# B&R Automation Studio project 305841_E00002_0 (part 5)

#### ActionMotionFbs.st
```iecst
(********************************************************************
 * COPYRIGHT -- General Atomics
 ********************************************************************
 * Program: AxisStateMachine
 * File: ActionMoveVel.st
 * Author: Administrator
 * Created: January 22, 2014
 ********************************************************************
 * Implementation of program AxisStateMachine
 ********************************************************************)

ACTION ActionCallMotionFunctions:
  ActionRangeCheckMoveParams;
  ActionMpAxisBasic;
  ActionReadDrivePos;
  ActionCamInOut;
  ActionGearInOut;
  ActionOffsetShift;
  ActionPhaseShift;
END_ACTION

ACTION ActionRangeCheckMoveParams:
  // Range checks position, velocity, accel & Decel

  // Make sure min/max values are not exceeded for position, velocity, accel, and decel.
  // Clamp if necessary.

  // Position
  ax.MoveParameters.Position := MIN(axPositionLimits.PositionLimitPos, MAX(axPositionLimits.PositionLimitNeg, ax.MoveParameters.Position));

  // Velocity
  ax.MoveParameters.Velocity := MIN(ax.MoveParameters.VelocityMax, MAX(ax.MoveParameters.VelocityMin, ax.MoveParameters.Velocity));

  // Accel and decel
  ax.MoveParameters.Acceleration := MIN(ax.MoveParameters.AccelMax, MAX(ax.MoveParameters.AccelMin, ax.MoveParameters.Acceleration));
  ax.MoveParameters.Deceleration := MIN(ax.MoveParameters.DecelMax, MAX(ax.MoveParameters.DecelMin, ax.MoveParameters.Deceleration));

END_ACTION

ACTION ActionMpAxisBasic:
  // 1) Assume velocity, accel & Decel have been range checked
  // 2) Packs the sMot_MoveParameters into a local axisBasicParamsStructure
  // 3) Detects parameter changes and manages the Update and UpdateDone bits
  // 4) Sets the fb command bits based on the axis sMot_AxisCommands structure
  // 5) Runs the fbMpAxisBasic funciton block
  // 6) Updates the axis structure with the status and axis info coming back from the fb

  // The execution behavior is determined by the inputs set elsewhere
  // in particular the sMot_AxisCommands XxxxCmd bits,
  // and the values in sMot_MoveParameters structure

  // Axis reference set in init routine

  // Only enable the fb if the axis is not set to be ignored
  // TODO: Different check needed? Not sure how to tell if an axis reference is not set
  // It would be nice to check ax.fbMpAxisBasic.MpLink <> 0 for example, but this is a structure not an address
  IF NOT ax.Ignore AND ax.AxisNo <> 0 THEN
    ax.fbMpAxisBasic.Enable := TRUE;
  ELSE
    ax.fbMpAxisBasic.Enable := FALSE;
  END_IF;

  // Load the parameters from the sMot_MoveParameter structure into
  // local structure variables used for the fb
  fctPackMpAxisBasicParams(_I_UdtParams:= ADR(ax.MoveParameters), _IO_MpParams := axisBasicParams);

  // To allow move parameter changes to take effect without having to stop,
  // detect a difference between the desired parameters and the previous values.
  // If they are different, then set the update bit until the UpdateDone bit is set.
  // NOTE: This fb manages the ax.fbMpAxisCoupling.Update request and monitors the .UpdateDone bit
  // Use the .UpdateCouplingParams bit in the command structure if the application needs to control
  // when to trigger the update. If parameters need to be set in possibly different areas of the software,
  // and all the updates should take place at once, the update fb is called conditionally. The
  // checked bit can be set high so it is called all the time if the checked bit is not managed.
  ax.Commands.UpdateMoveParams:= TRUE;
  IF ax.Commands.UpdateMoveParams THEN
    ax.fbUpdateBFbParams(_IO_MpParams := axisBasicParams);
    ax.Commands.UpdateMoveParams := FALSE;
  END_IF;

  // TODO: Enforce move permissives

  // Use the commands from the axis structue
  ax.fbMpAxisBasic.ErrorReset := ax.Commands.DriveResetCmd;
  ax.fbMpAxisBasic.Power := ax.Commands.EnableCmd;
  ax.fbMpAxisBasic.Home := ax.Commands.HomeCmd;
  // There is no specific jog cmd. Use Move Velocity instead.
  ax.fbMpAxisBasic.MoveVelocity := ax.Commands.MoveVelocityCmd OR ax.Commands.MoveJogCmd;
  ax.fbMpAxisBasic.MoveAbsolute := ax.Commands.MoveAbsoluteCmd;
  ax.fbMpAxisBasic.MoveAdditive := ax.Commands.MoveRelativeCmd;
  ax.fbMpAxisBasic.Stop := ax.Commands.StopCmd;
  ax.fbMpAxisBasic.JogPositive := ax.Commands.MoveJogPositiveCmd;
  ax.fbMpAxisBasic.JogNegative := ax.Commands.MoveJogNegativeCmd;
  ax.fbMpAxisBasic.LimitLoad := ax.MoveParameters.EnableTorqueLimit;
  ax.fbMpAxisBasic.ReleaseBrake := ax.Commands.ReleaseBrakeCmd;
  ax.fbMpAxisBasic.AutoTune := FALSE; // TODO
  ax.fbMpAxisBasic.Simulate := FALSE; // TODO

  // Call the fb
  ax.fbMpAxisBasic();

  // Update the axis status structure
  ax.Status.Position := ax.fbMpAxisBasic.Position;
  ax.Status.Velocity := ax.fbMpAxisBasic.Velocity;
  ax.Status.IsPoweredOn := ax.fbMpAxisBasic.PowerOn;
  ax.Status.IsHomed := ax.fbMpAxisBasic.IsHomed;
  ax.Status.IsInVelocity := ax.fbMpAxisBasic.InVelocity;
  ax.Status.IsInPosition := ax.fbMpAxisBasic.InPosition;
  ax.Status.IsMoveActive := ax.fbMpAxisBasic.MoveActive;
  ax.Status.IsMoveDone := ax.fbMpAxisBasic.MoveDone;
  ax.Status.IsStopped := ax.fbMpAxisBasic.Stopped;
  ax.Status.IsTorqueLimitReady := ax.fbMpAxisBasic.LimitLoadReady;
  ax.Status.IsBrakeManuallyReleased := ax.fbMpAxisBasic.BrakeReleased;

  // Now load the sMot_AxisStatus structure with the data returned from the fb
  fctGetMpAxisInfo(_I_MpInfo := ADR(ax.fbMpAxisBasic.Info), _IO_UdtStatus := ax.Status);

  // Calculate special (algorithmic) positions
  CalcSpecialPositions;

  // Now that the status of this axis is known, copy it to the other axes slave status
  // area if this axis is specified as a slave.
  CopySlaveStatusToMaster;

END_ACTION

ACTION ActionReadDrivePos:
  // Read the drive position. As opposed to the position value coming from MpAxisBasic,
  // the drive position allows different position sources to be specified, but it also
  // allows can provide the position that does not have a MOD applied in the periodic case.
  // This is helpful to assess long moves on periodic axes (e.g. 1000 degree move on a
  // 360 degree periodic axis).
  // Only execute the read position fb if the axis number has been set,
  // the axis is not ignored.
  IF NOT ax.Ignore AND ax.AxisNo <> AD_UNKNOWN THEN
    // Axis is in play. Go get some of that position ...
    // Set the source, enable the fb
    ax.fbReadDrivePos.ValueSource := mcVALUE_ACTUAL_AXIS_UNITS;
    ax.fbReadDrivePos.Enable := TRUE;
  ELSE
    // axis should be ignored
    // keep the enable low
    ax.fbReadDrivePos.Enable := FALSE;
  END_IF;

  // Fb should be set up. Call 'er
  ax.fbReadDrivePos();

  // If fb has been enabled and is valid and error , get the drive position. Otherwise
  // use the sentinel value
  IF ax.fbReadDrivePos.Enable AND ax.fbReadDrivePos.Valid AND NOT ax.fbReadDrivePos.Error THEN
    ax.Status.DrivePosition := ax.fbReadDrivePos.CyclicPosition;
  ELSE
    ax.Status.DrivePosition := INVALID_SENTINEL_LREAL;
  END_IF;

END_ACTION

ACTION ActionCamInOut:
  // Execute the cam in or cam out fbs based on the CamIn/Out requests
  // The fbs are edge triggered, and the requests are cleared once serviced.
  // If the caming params change, another request must be made.
  // TODO: Is cam out and another cam in needed if params change?

  // Only execute the cam in fb if the axis number has been set,
  // the slave axis number has been set, and neither is set to be ignored,
  // and it is requested.
  IF ax.Ignore OR ax.AxisNo = AD_UNKNOWN OR
       ax.CouplingParameters.SlaveAxisNo = AD_UNKNOWN OR
       axes[ax.CouplingParameters.SlaveAxisNo].Ignore THEN
    // slave or master should be ignored
    // keep the requests and executes low
    ax.CouplingParameters.CamInReq := FALSE;
    ax.CouplingParameters.CamOutReq := FALSE;
    ax.fbCamIn.Execute := FALSE;
    ax.fbCamOut.Execute := FALSE;
  ELSIF ax.CouplingParameters.CamInReq THEN
    // CamIn request is made.
    // Clear the req so a future rising edge can be seen
    ax.CouplingParameters.CamInReq := FALSE;
    // Make sure the CamOut req and execute is clear
    ax.CouplingParameters.CamOutReq := FALSE;
    ax.fbCamOut.Execute := FALSE;
    // Load the cam in params, then set the execute input (edge triggered fb)
    ax.fbCamIn.MasterOffset := ax.CouplingParameters.CamMasterOffset;
    ax.fbCamIn.SlaveOffset := ax.CouplingParameters.CamSlaveOffset;
    ax.fbCamIn.MasterScaling := ax.CouplingParameters.CamScalingMaster;
    ax.fbCamIn.SlaveScaling := ax.CouplingParameters.CamScalingSlave;
    ax.fbCamIn.StartMode := ax.CouplingParameters.CamStartMode;
    ax.fbCamIn.MasterValueSource := ax.CouplingParameters.CamMasterValueSource;
    ax.fbCamIn.CamID := ax.CouplingParameters.CamId;
    ax.fbCamIn.BufferMode := ax.CouplingParameters.CamBufferMode; // only mcAborting currently supported
    ax.fbCamIn.AdvancedParameters.Periodic := ax.CouplingParameters.CamIsPeriodic;
    ax.fbCamIn.AdvancedParameters.Velocity := 0.0; // disable, use (slave?) axis max vel
    ax.fbCamIn.AdvancedParameters.Acceleration := 0.0; // disable, use (slave?) axis max accel
    ax.fbCamIn.AdvancedParameters.Deceleration := 0.0; // disable, use (slave?) axis max decel
    ax.fbCamIn.AdvancedParameters.Jerk := 0.0; // only non-zero if using McProfGen
    ax.fbCamIn.Execute := TRUE; // fb looks for a rising edge
  ELSIF ax.CouplingParameters.CamOutReq THEN
    // Clear the req so a future rising edge can be seen
    ax.CouplingParameters.CamOutReq := FALSE;
    // Make sure the GearIn req and execute is clear
    ax.CouplingParameters.CamInReq := FALSE;
    ax.fbCamIn.Execute := FALSE;
    // Load the cam out params, then set the execute input (edge triggered fb)
    ax.fbCamOut.Jerk := 0.0; // only non-zero if using McProfGen
    ax.fbCamOut.Execute := TRUE;
  END_IF;

  // Call the cam in and cam out fbs.
  ax.fbCamIn();
  ax.fbCamOut();
  // Clear the exuecute bits. The fbs are edge triggerd, and would have been seen by the above call.
  ax.fbCamIn.Execute := FALSE;
  ax.fbCamOut.Execute := FALSE;

  // Update the axis status structure
  IF NOT ax.fbCamIn.Error THEN
    ax.Status.IsCamInSync := ax.fbCamIn.InSync;
    ax.Status.IsCamEndOfProfile := ax.fbCamIn.EndOfProfile;
    ax.Status.CamStatus := ax.fbCamIn.Status;
  ELSE
    ax.Status.IsCamInSync := FALSE;
    ax.Status.IsCamEndOfProfile := FALSE;
    ax.Status.CamStatus := mcCAM_STATUS_PREPARING_MOVE; // 0 value, but don't have a good choice for "not active"
  END_IF;

END_ACTION

ACTION ActionGearInOut:
  // Execute the gear in or gear out fbs based on the GearIn/Out requests
  // The fbs are edge triggered, and the requests are cleared once serviced.
  // If the gearing params change, another request must be made.

  // Only execute the gear in fb if the axis number has been set,
  // the slave axis number has been set, and neither is set to be ignored,
  // and it is requested.
  IF ax.Ignore OR ax.AxisNo = AD_UNKNOWN OR
       ax.CouplingParameters.SlaveAxisNo = AD_UNKNOWN OR
       axes[ax.CouplingParameters.SlaveAxisNo].Ignore THEN
    // slave or master should be ignored
    // keep the requests and executes low
    ax.CouplingParameters.GearInReq := FALSE;
    ax.CouplingParameters.GearOutReq := FALSE;
    ax.fbGearIn.Execute := FALSE;
    ax.fbGearOut.Execute := FALSE;
  ELSIF ax.CouplingParameters.GearInReq THEN
    // GearIn request is made.
    // Clear the req so a future rising edge can be seen
    ax.CouplingParameters.GearInReq := FALSE;
    // Make sure the GearOut req and execute is clear
    ax.CouplingParameters.GearOutReq := FALSE;
    ax.fbGearOut.Execute := FALSE;
    // Load the gear in params, then set the execute input (edge triggered fb)
    ax.fbGearIn.RatioNumerator := ax.CouplingParameters.GearInRatioNumerator;
    ax.fbGearIn.RatioDenominator := ax.CouplingParameters.GearInRatioDenominator;
    ax.fbGearIn.MasterValueSource := ax.CouplingParameters.GearInMasterValueSource;
    ax.fbGearIn.Acceleration := ax.CouplingParameters.ShiftAccelerationMax;
    ax.fbGearIn.Deceleration := ax.CouplingParameters.ShiftDecelerationMax;
    ax.fbGearIn.Jerk := ax.CouplingParameters.ShiftJerk; // only non-zero if using McProfGen
    ax.fbGearIn.BufferMode := ax.CouplingParameters.GearInBufferMode; // onlly mcAborting currently supported
    ax.fbGearIn.AdvancedParameters.MasterMaxVelocity := ax.CouplingParameters.ShiftProfileBaseMaxVelocity;
    ax.fbGearIn.Execute := TRUE; // fb looks for a rising edge
  ELSIF ax.CouplingParameters.GearOutReq THEN
    // Clear the req so a future rising edge can be seen
    ax.CouplingParameters.GearOutReq := FALSE;
    // Make sure the GearIn req and execute is clear
    ax.CouplingParameters.GearInReq := FALSE;
    ax.fbGearIn.Execute := FALSE;
    // Load the gear out params, then set the execute input (edge triggered fb)
    ax.fbGearOut.Jerk := 0.0; // only non-zero if using McProfGen
    ax.fbGearOut.Execute := TRUE;
  END_IF;

  // Call the gear in and gear out fbs.
  ax.fbGearIn();
  ax.fbGearOut();
  // Clear the exuecute bits. The fbs are edge triggerd, and would have been seen by the above call.
  ax.fbGearIn.Execute := FALSE;
  ax.fbGearOut.Execute := FALSE;

  // Update the axis status structure.
  // Derrive InCompensation -- Active but not in sync
  IF ax.fbGearIn.Active AND NOT ax.fbGearIn.Error THEN
    // If gear in is active, it is either in sync or in compensation
    ax.Status.IsGearInSync := ax.fbGearIn.InGear;
    ax.Status.IsGearInCompensation := NOT ax.fbGearIn.InGear;
  ELSE
    ax.Status.IsGearInSync := FALSE;
    ax.Status.IsGearInCompensation := FALSE;
  END_IF;

END_ACTION

ACTION ActionOffsetShift:
  // Execute the offset shift fb based on the offset shift request.
  // The fb has a level sensitive enable and an edge triggered StartShift input.
  // NOTE: Either by design or because of a bug, the AdvancedParameters.ProfileBase
  // seems to be evaluated based on Enable going high. Changes made to the ProfileBase,
  // after enable going high but before StartShift input going high are ignored.
  // If the shift params change, another request must be made.
  // A shift cannot be stopped once started without halting or some oher means of stopping
  // the axes outside the scope of the shift fb.

  // Since triggering an offset while another shift is in progress triggers an error,
  // the request, enable, and start shift are only cleared once the shift is finished,
  // or the fb is invalid or in error

  // Only execute the offset shift fb if the axis number has been set,
  // the slave axis number has been set, and neither is set to be ignored
  IF ax.Ignore OR ax.AxisNo = AD_UNKNOWN OR
    ax.CouplingParameters.SlaveAxisNo = AD_UNKNOWN OR
    axes[ax.CouplingParameters.SlaveAxisNo].Ignore THEN
    // slave or master should be ignored, or slave is not set, or
    // master is not powered.  Keep the request, enable, and startshift low
    ax.CouplingParameters.OffsetShiftReq := FALSE;
    ax.fbOffsetShift.Enable := FALSE;
    ax.fbOffsetShift.StartShift := FALSE;
  ELSIF ax.CouplingParameters.OffsetShiftReq AND NOT ax.fbOffsetShift.Enable THEN
    // Offset Shift request is made.
    // Set the fb params so a start shift can act on them. Set them
    // before bringing enable high because the profile base param(s) seem to
    // need to be set before the StartShift input is raised.
    ax.fbOffsetShift.OffsetShift := ax.CouplingParameters.Shift;
    ax.fbOffsetShift.Velocity := ax.CouplingParameters.ShiftVelocityMax;
    ax.fbOffsetShift.Acceleration := ax.CouplingParameters.ShiftAccelerationMax;
    ax.fbOffsetShift.AdvancedParameters.ShiftMode := ax.CouplingParameters.ShiftMode;
    ax.fbOffsetShift.AdvancedParameters.ProfileBase := ax.CouplingParameters.ShiftProfileBase;
    ax.fbOffsetShift.AdvancedParameters.ProfileBaseMaxVelocity := ax.CouplingParameters.ShiftProfileBaseMaxVelocity;
    ax.fbOffsetShift.AdvancedParameters.DistanceParameters.ProfileDistance := ax.CouplingParameters.ShiftProfileDistance;
    ax.fbOffsetShift.AdvancedParameters.ZoneParameters.StartPosition := ax.CouplingParameters.ShiftZoneStartPosition;
    ax.fbOffsetShift.AdvancedParameters.ZoneParameters.EndPosition := ax.CouplingParameters.ShiftZoneEndPosition;
    ax.fbOffsetShift.AdvancedParameters.ZoneParameters.Period := ax.CouplingParameters.ShiftZonePeriod;
    ax.fbOffsetShift.AdvancedParameters.ShiftAlternativeValueSource := mcALT_VALUE_NOT_USED;
    // Enable the fb so we can look for a valid before starting the shift.
    ax.fbOffsetShift.Enable := TRUE;
  ELSIF ax.CouplingParameters.OffsetShiftReq AND ax.fbOffsetShift.Enable AND
    NOT ax.fbOffsetShift.StartShift AND ax.fbOffsetShift.Valid AND NOT ax.fbOffsetShift.Error THEN
    // fb is enabled and valid and not in error, but not started yet.
    // Start the shift on the edge triggered StartShift input.
    ax.fbOffsetShift.StartShift := TRUE;
  ELSIF ax.CouplingParameters.OffsetShiftReq AND ax.fbOffsetShift.Enable AND ax.fbOffsetShift.Error THEN
    // fb is enabled but in error. Clear the request, enable, and make sure the start shift stays low
    ax.CouplingParameters.OffsetShiftReq := FALSE;
    ax.fbOffsetShift.Enable := FALSE;
    ax.fbOffsetShift.StartShift := FALSE;
  ELSIF ax.CouplingParameters.OffsetShiftReq AND ax.fbOffsetShift.Valid AND ax.fbOffsetShift.StartShift AND
    NOT ax.fbOffsetShift.ShiftAttained THEN
    // Shift was triggered, but isn't done yet.
    // Update the axis status structure
    ax.Status.IsCoordOffsetShiftAttained := FALSE;
    ax.Status.IsCoordOffsetShiftStarted := ax.fbOffsetShift.ShiftStarted;
    ax.Status.CoordActualOffsetShift := ax.fbOffsetShift.ActualOffsetShift;
  ELSIF ax.CouplingParameters.OffsetShiftReq AND ax.fbOffsetShift.Valid AND ax.fbOffsetShift.StartShift AND
    ax.fbOffsetShift.ShiftAttained THEN
    // Shift was triggered, and is now done.
    // Update the axis status structure
    ax.Status.IsCoordOffsetShiftAttained := ax.fbOffsetShift.ShiftAttained;
    ax.Status.IsCoordOffsetShiftStarted := FALSE;
    ax.Status.CoordActualOffsetShift := ax.fbOffsetShift.ActualOffsetShift;
    // Clear the request, enable, and start shift.
    // Clearing the original request at the end prevents another request from triggering a shift while
    // a shift is in progress, but also allows another request to be triggered once done.
    ax.CouplingParameters.OffsetShiftReq := FALSE;
    ax.fbOffsetShift.Enable := FALSE;
    ax.fbOffsetShift.StartShift := FALSE;
  END_IF;

  // Call the offset shift fb.
  ax.fbOffsetShift();

END_ACTION

ACTION ActionPhaseShift:
  // Execute the phase shift fb based on the phase shift request.
  // The fb has a level sensitive enable and an edge triggered StartShift input.
  // NOTE: Either by design or because of a bug, the AdvancedParameters.ProfileBase
  // seems to be evaluated based on Enable going high. Changes made to the ProfileBase,
  // after enable going high but before StartShift input going high are ignored.
  // If the shift params change, another request must be made.
  // A shift cannot be stopped once started without halting or some oher means of stopping
  // the axes outside the scope of the shift fb.

  // Since triggering phase shift while another shift is in progress triggers an error,
  // the request, enable, and start shift are only cleared once the shift is finished,
  // or the fb is invalid or in error

  // Only execute the phase shift fb if the axis number has been set,
  // the slave axis number has been set, and neither is set to be ignored
  IF ax.Ignore OR ax.AxisNo = AD_UNKNOWN OR
    ax.CouplingParameters.SlaveAxisNo = AD_UNKNOWN OR
    axes[ax.CouplingParameters.SlaveAxisNo].Ignore THEN
    // slave or master should be ignored, or slave is not set, or
    // master is not powered.  Keep the request, enable, and startshift low
    ax.CouplingParameters.PhaseShiftReq := FALSE;
    ax.fbPhaseShift.Enable := FALSE;
    ax.fbPhaseShift.StartShift := FALSE;
  ELSIF ax.CouplingParameters.PhaseShiftReq AND NOT ax.fbPhaseShift.Enable THEN
    // Phase Shift request is made.
    // Set the fb params so a start shift can act on them. Set them
    // before bringing enable high because the profile base param(s) seem to
    // need to be set before the StartShift input is raised.
    ax.fbPhaseShift.PhaseShift := ax.CouplingParameters.Shift;
    ax.fbPhaseShift.Velocity := ax.CouplingParameters.ShiftVelocityMax;
    ax.fbPhaseShift.Acceleration := ax.CouplingParameters.ShiftAccelerationMax;
    ax.fbPhaseShift.AdvancedParameters.ShiftMode := ax.CouplingParameters.ShiftMode;
    ax.fbPhaseShift.AdvancedParameters.ProfileBase := ax.CouplingParameters.ShiftProfileBase;
    ax.fbPhaseShift.AdvancedParameters.ProfileBaseMaxVelocity := ax.CouplingParameters.ShiftProfileBaseMaxVelocity;
    ax.fbPhaseShift.AdvancedParameters.DistanceParameters.ProfileDistance := ax.CouplingParameters.ShiftProfileDistance;
    ax.fbPhaseShift.AdvancedParameters.ZoneParameters.StartPosition := ax.CouplingParameters.ShiftZoneStartPosition;
    ax.fbPhaseShift.AdvancedParameters.ZoneParameters.EndPosition := ax.CouplingParameters.ShiftZoneEndPosition;
    ax.fbPhaseShift.AdvancedParameters.ZoneParameters.Period := ax.CouplingParameters.ShiftZonePeriod;
    ax.fbPhaseShift.AdvancedParameters.ShiftAlternativeValueSource := mcALT_VALUE_NOT_USED;
    // Enable the fb so we can look for a valid before starting the shift.
    ax.fbPhaseShift.Enable := TRUE;
  ELSIF ax.CouplingParameters.PhaseShiftReq AND ax.fbPhaseShift.Enable AND
    NOT ax.fbPhaseShift.StartShift AND ax.fbPhaseShift.Valid AND NOT ax.fbPhaseShift.Error THEN
    // fb is enabled and valid and not in error, but not started yet.
    // Start the shift on the edge triggered StartShift input.
    ax.fbPhaseShift.StartShift := TRUE;
  ELSIF ax.CouplingParameters.PhaseShiftReq AND ax.fbPhaseShift.Enable AND ax.fbPhaseShift.Error THEN
    // fb is enabled but in error. Clear the request, enable, and make sure the start shift stays low
    ax.CouplingParameters.PhaseShiftReq := FALSE;
    ax.fbPhaseShift.Enable := FALSE;
    ax.fbPhaseShift.StartShift := FALSE;
  ELSIF ax.CouplingParameters.PhaseShiftReq AND ax.fbPhaseShift.Valid AND ax.fbPhaseShift.StartShift AND
    NOT ax.fbPhaseShift.ShiftAttained THEN
    // Shift was triggered, but isn't done yet.
    // Update the axis status structure
    ax.Status.IsCoordPhaseShiftAttained := FALSE;
    ax.Status.IsCoordPhaseShiftStarted := ax.fbPhaseShift.ShiftStarted;
    ax.Status.CoordActualPhaseShift := ax.fbPhaseShift.ActualPhaseShift;
  ELSIF ax.CouplingParameters.PhaseShiftReq AND ax.fbPhaseShift.Valid AND ax.fbPhaseShift.StartShift AND
    ax.fbPhaseShift.ShiftAttained THEN
    // Shift was triggered, and is now done.
    // Update the axis status structure
    ax.Status.IsCoordPhaseShiftAttained := ax.fbPhaseShift.ShiftAttained;
    ax.Status.IsCoordPhaseShiftStarted := FALSE;
    ax.Status.CoordActualPhaseShift := ax.fbPhaseShift.ActualPhaseShift;
    // Clear the request, enable, and start shift.
    // Clearing the original request at the end prevents another request from triggering a shift while
    // a shift is in progress, but also allows another request to be triggered once done.
    ax.CouplingParameters.PhaseShiftReq := FALSE;
    ax.fbPhaseShift.Enable := FALSE;
    ax.fbPhaseShift.StartShift := FALSE;
  END_IF;

  // Call the phase shift fb.
  ax.fbPhaseShift();

END_ACTION

ACTION CopySlaveStatusToMaster :
  // If this axis number is a slave to another axis, then copy this axis
  // status to the master axis structure. This is a convenience
  // so the HMI for example, only needs to look in one structure (the master) and
  // can access the slave status.

  // Loop thru the axes. If the axis of index has this axis specified as a slave axis,
  // copy this axis status to the axis of index slave status.
  // Axis 0 is a dummy axis, so it can be skipped.
  FOR axIdx := 1 TO AXIS_COUNT DO
    IF axes[axIdx].CouplingParameters.SlaveAxisNo = AXIS_NO THEN
      // This axis is a slave to the axis referenced by axIdx.
      // Copy this axis status to the indexed axis slave status
      fctCopyAxisStatus(_I_SrcStatus := ADR(ax.Status), _I_DestStatus := ADR(axes[axIdx].StatusSlave));
    END_IF;
  END_FOR;
END_ACTION
```

- ActionMotionFbs.st.bak (not shown)

#### AxSMInit.st
```iecst
PROGRAM _INIT
  // set ax pointer to the element of the global sMot_Axis array
  ax ACCESS ADR(axes[AXIS_NO]);

  // set the position limits to point to the global permanent variable
  axPositionLimits ACCESS ADR(gr_AxisPositionLimits[AXIS_NO]);

  // Set the axis number and clear the ignore bit
  ax.AxisNo:= AXIS_NO;

  // **** These settings need to be reviewed/set for each axis
  ax.CouplingParameters.SlaveAxisNo := DINT_TO_USINT(AD_INNER_ECCENTRIC); // Inner axis will be the slave to the outer axis
  ax.Ignore := FALSE;
  ax.isAxisEndless := TRUE;
  ax.isAxisVirtual := FALSE;
  ax.isAxisInverter := FALSE;

  // Point to the mappMotion axis, and a slave if there is one
  ax.AxisObj := gAxOutE; // mappMotion axis -- see mappMotion in cfg view
  ax.SlaveAxisObj := gAxInE; // no slave for the Z Axis

  // Set the restore pos check fb
  ax.fbCheckRestorePos.Axis := ADR(ax.AxisObj);
  ax.fbCheckRestorePos.DataAddress := ADR(gr_AxOutERestorePos); // Set this per axis

  // Load the min/max velocity and accel/decel from constants
  ax.MoveParameters.AccelMin := 0.001; // TODO: Not sure of a good value, but it should not be zero.
  ax.MoveParameters.AccelMax:= AXIS_OUTE_MAX_ACCEL;
  ax.MoveParameters.DecelMin := 0.001; // TODO:Not sure of a good value, but it should not be zero.
  ax.MoveParameters.DecelMax:= AXIS_OUTE_MAX_DECEL;
  ax.MoveParameters.VelocityMin := -1.0 * AXIS_OUTE_MAX_VELOCITY;
  ax.MoveParameters.VelocityMax := AXIS_OUTE_MAX_VELOCITY;

  // **** The settings below don't normally need to be altered

  // set the fb axis references
  ax.fbMpAxisBasic.MpLink := ADR(ax.AxisObj);
  ax.fbReadDrivePos.Axis:= ADR(ax.AxisObj);
  ax.fbGearIn.Master := ADR(ax.AxisObj);
  ax.fbGearIn.Slave := ADR(ax.SlaveAxisObj);
  ax.fbGearOut.Slave := ADR(ax.SlaveAxisObj);
  ax.fbOffsetShift.Slave := ADR(ax.SlaveAxisObj);
  ax.fbPhaseShift.Slave := ADR(ax.SlaveAxisObj);
  ax.fbCamIn.Master := ADR(ax.AxisObj);
  ax.fbCamIn.Slave := ADR(ax.SlaveAxisObj);
  ax.fbCamOut.Slave := ADR(ax.SlaveAxisObj);
  ax.fbUpdateBFbParams._I_Axis := ADR(ax);

  // Set fb reference to local variables
  ax.fbMpAxisBasic.Parameters := ADR(axisBasicParams);

  // Set previous values for motion parameters so changes can be detected
  ax.MoveParametersPrev := ax.MoveParameters;

  // Clear commands and requests
  fctClearMotionCommands(_I_CmdMask := MACM_NOMASK, _IO_Commands := ax.Commands);
  fctClearMotionRequests(_I_ReqMask := MACM_NOMASK, _IO_Commands := ax.Commands);

  // set the move not allowed flag
  ax.Commands.MoveNotAllowed:= TRUE;

  // Set the most primitive status. If the axis is valid, the
  // full status will be updated later once comms is established, and the drive status is updated via MpAxisBasic
  ax.Status.IsCommuncationReady := FALSE;
  ax.Status.IsReadyToPowerOn := FALSE;

END_PROGRAM
```

### Program Logical/PlcLogic/axInE/axInESM (IEC) - Axis State Machine

#### AxSM.var
```iecst
(********************************************************************
 * COPYRIGHT -- General Atomics
 ********************************************************************
 * Program: AFtInSM
 * File: AFtInSM.var
 * Author: Administrator
 * Created: July 16, 2014
 ********************************************************************
 * Local variables of program AFtInSM
 ********************************************************************)
VAR CONSTANT
  (* axis number is per eAXIS_DESIGNATION *)
  (*
    AD_UNKNOWN := 0,
    AD_SPINDLE := 1,
    AD_OUTER_ECCENTRIC := 2,
    AD_INNER_ECCENTRIC := 3,
    AD_Z := 4,
    derrived axes
    AD_X := 5,
    AD_Y := 6,
    virual axes
    AD_HANDWHEEL := 7
  *)

  (* same info but different data types for convenience *)
  AXIS_NO : USINT := AD_INNER_ECCENTRIC; (* USINT so it can be used as an array index *)
  AXIS_DESIGNATION : eAXIS_DESIGNATION := AD_INNER_ECCENTRIC;

  END_VAR

  VAR
  ax : REFERENCE TO sMot_Axis;
  axPositionLimits : REFERENCE TO sMot_PositionLimits;
  axIdx : DINT; (* axis index *)
  inSyncSlave : BOOL := FALSE;
  axDummySlave : McAxisType;
	axisBasicParams : MpAxisBasicParType; (* local version -- used to make address referencing easier *)
	axisCouplingParams : MpAxisCouplingParType;
  tmrStepTO : TON; (* Step TO timer *)
  reqMask : DINT := MACM_NOMASK; (* request mask *)
  cmdMask : DINT := MACM_NOMASK; (* command mask *)
  tmrDriveReset : TON; (* auto issue drive reset while invalid also used to force minimum time in error states *)
	tmrModeMismatch : TON; (* mode mismatch timer *)
	tmrHomeMinimum : TON; (* force Home cmd to be present before transitioning *)
END_VAR
```

#### ActionAxisSpecific.st
```iecst
ACTION CalcSpecialPositions :
  // If there is an algorithm needed for calculating a different position, it can be done here
  // If not, just use the axis position.

  // CalculatedPosition1
  // Calculate the inner position relative to the outer position, in degrees.
  // This assumes the zero/home position of both the Outer and Inner axes was set to zero when
  // the index lines are lined up with each other.
  // Calculated Position = Inner Pos - Outer Pos.
  // Make the result be +/- 180 degrees:
  // If I-O > 180 :  Calc Pos = Result - 360
  // If I-O < -180 : Calc Pos = Result + 360
  // The fctAziDiff function in GAMath library does this (pos A - pos B)

  IF NOT axes[AD_INNER_ECCENTRIC].Status.IsHomed OR NOT axes[AD_OUTER_ECCENTRIC].Status.IsHomed THEN
    // Inner and/or outer axis is not homed.
    // Use the sentinel value for the calculated positions.
    ax.Status.CalculatedPosition1 := INVALID_SENTINEL_REAL;
  ELSE
    // Both the inner and outer axes are referenced.
    // Calc the difference between them. I - O
    ax.Status.CalculatedPosition1 := fctAziDiff(
    _I_PosA :=  ax.Status.Position,
    _I_PosB := axes[AD_OUTER_ECCENTRIC].Status.Position);
  END_IF;

  ax.Status.CalculatedPosition2 := ax.Status.Position;
  ax.Status.CalculatedPosition3 := ax.Status.Position;

END_ACTION
```

#### ActionMotionFbs.st
```iecst
(********************************************************************
 * COPYRIGHT -- General Atomics
 ********************************************************************
 * Program: AxisStateMachine
 * File: ActionMoveVel.st
 * Author: Administrator
 * Created: January 22, 2014
 ********************************************************************
 * Implementation of program AxisStateMachine
 ********************************************************************)

ACTION ActionCallMotionFunctions:
  ActionMpAxisBasic;
  ActionMpAxisCoupling;
END_ACTION

ACTION ActionMpAxisBasic:
  // 1) Range checks position, velocity, accel & Decel
  // 2) Packs the sMot_MoveParameters into a local axisBasicParamsStructure
  // 3) Detects parameter changes and manages the Update and UpdateDone bits
  // 4) Sets the fb command bits based on the axis sMot_AxisCommands structure
  // 5) Runs the fbMpAxisBasic funciton block
  // 6) Updates the axis structure with the status and axis info coming back from the fb

  // Make sure min/max values are not exceeded for position, velocity, accel, and decel.
  // Clamp if necessary

  // Position
  IF ax.MoveParameters.Position >  axPositionLimits.PositionLimitPos THEN
    ax.MoveParameters.Position :=  axPositionLimits.PositionLimitPos;
  END_IF;
  IF ax.MoveParameters.Position <  axPositionLimits.PositionLimitNeg THEN
    ax.MoveParameters.Position :=  axPositionLimits.PositionLimitNeg;
  END_IF;

  // Velocity
  IF ax.MoveParameters.Velocity > ax.MoveParameters.VelocityMax THEN
    ax.MoveParameters.Velocity := ax.MoveParameters.VelocityMax;
  END_IF;
  IF ax.MoveParameters.Velocity < ax.MoveParameters.VelocityMin THEN
    ax.MoveParameters.Velocity := ax.MoveParameters.VelocityMin;
  END_IF;

  // Accel and decel
  IF ax.MoveParameters.Acceleration > ax.MoveParameters.AccelMax THEN
    ax.MoveParameters.Acceleration := ax.MoveParameters.AccelMax;
  END_IF;
  IF ax.MoveParameters.Acceleration < ax.MoveParameters.AccelMin THEN
    ax.MoveParameters.Acceleration := ax.MoveParameters.AccelMin;
  END_IF;

  IF ax.MoveParameters.Deceleration > ax.MoveParameters.DecelMax THEN
    ax.MoveParameters.Deceleration := ax.MoveParameters.DecelMax;
  END_IF;
  IF ax.MoveParameters.Deceleration < ax.MoveParameters.DecelMin THEN
    ax.MoveParameters.Deceleration := ax.MoveParameters.DecelMin;
  END_IF;

  // The execution behavior is determined by the inputs set elsewhere
  // in particular the sMot_AxisCommands XxxxCmd bits,
  // and the values in sMot_MoveParameters structure

  // Axis reference set in init routine

  // Only enable the fb if the axis is not set to be ignored
  // TODO: Different check needed? Not sure how to tell if an axis reference is not set
  // It would be nice to check ax.fbMpAxisBasic.MpLink <> 0 for example, but this is a structure not an address
  IF NOT ax.Ignore AND ax.AxisNo <> 0 THEN
    ax.fbMpAxisBasic.Enable := TRUE;
  ELSE
    ax.fbMpAxisBasic.Enable := FALSE;
  END_IF;

  // Load the parameters from the sMot_MoveParameter structure into
  // local structure variables used for the fb
  fctPackMpAxisBasicParams(_I_UdtParams:= ADR(ax.MoveParameters), _IO_MpParams := axisBasicParams);

  // To allow move parameter changes to take effect without having to stop,
  // detect a difference between the desired parameters and the previous values.
  // If they are different, then set the update bit until the UpdateDone bit is set.
  // NOTE: This fb manages the ax.fbMpAxisCoupling.Update request and monitors the .UpdateDone bit
  // Use the .UpdateCouplingParams bit in the command structure if the application needs to control
  // when to trigger the update. If parameters need to be set in possibly different areas of the software,
  // and all the updates should take place at once, the update fb is called conditionally. The
  // checked bit can be set high so it is called all the time if the checked bit is not managed.
  ax.Commands.UpdateMoveParams:= TRUE;
  IF ax.Commands.UpdateMoveParams THEN
    ax.fbUpdateBFbParams(_IO_MpParams := axisBasicParams);
    ax.Commands.UpdateMoveParams := FALSE;
  END_IF;

  // TODO: Enforce move permissives

  // Use the commands from the axis structue
  ax.fbMpAxisBasic.ErrorReset := ax.Commands.DriveResetCmd;
  ax.fbMpAxisBasic.Power := ax.Commands.EnableCmd;
  ax.fbMpAxisBasic.Home := ax.Commands.HomeCmd;
  // There is no specific jog cmd. Use Move Velocity instead.
  ax.fbMpAxisBasic.MoveVelocity := ax.Commands.MoveVelocityCmd OR ax.Commands.MoveJogCmd;
  ax.fbMpAxisBasic.MoveAbsolute := ax.Commands.MoveAbsoluteCmd;
  ax.fbMpAxisBasic.MoveAdditive := ax.Commands.MoveRelativeCmd;
  ax.fbMpAxisBasic.Stop := ax.Commands.StopCmd;
  ax.fbMpAxisBasic.JogPositive := ax.Commands.MoveJogPositiveCmd;
  ax.fbMpAxisBasic.JogNegative := ax.Commands.MoveJogNegativeCmd;
  ax.fbMpAxisBasic.LimitLoad := ax.MoveParameters.EnableTorqueLimit;
  ax.fbMpAxisBasic.ReleaseBrake := ax.Commands.ReleaseBrakeCmd;
  ax.fbMpAxisBasic.AutoTune := FALSE; // TODO
  ax.fbMpAxisBasic.Simulate := FALSE; // TODO

  // Call the fb
  ax.fbMpAxisBasic();

  // Update the fb status structure
  ax.statusFpMpAxisBasic.Active := ax.fbMpAxisBasic.Active;
  ax.statusFpMpAxisBasic.Error := ax.fbMpAxisBasic.Error;
  ax.statusFpMpAxisBasic.StatusId := ax.fbMpAxisBasic.StatusID;
  ax.statusFpMpAxisBasic.UpdateDone := ax.fbMpAxisBasic.UpdateDone;
  ax.statusFpMpAxisBasic.CommandBusy := ax.fbMpAxisBasic.CommandBusy;
  ax.statusFpMpAxisBasic.CommandAborted := ax.fbMpAxisBasic.CommandAborted;

  // Update the axis status structure
  ax.Status.Position := ax.fbMpAxisBasic.Position;
  ax.Status.Velocity := ax.fbMpAxisBasic.Velocity;
  ax.Status.IsPoweredOn := ax.fbMpAxisBasic.PowerOn;
  ax.Status.IsHomed := ax.fbMpAxisBasic.IsHomed;
  ax.Status.IsInVelocity := ax.fbMpAxisBasic.InVelocity;
  ax.Status.IsInPosition := ax.fbMpAxisBasic.InPosition;
  ax.Status.IsMoveActive := ax.fbMpAxisBasic.MoveActive;
  ax.Status.IsMoveDone := ax.fbMpAxisBasic.MoveDone;
  ax.Status.IsStopped := ax.fbMpAxisBasic.Stopped;
  ax.Status.IsTorqueLimitReady := ax.fbMpAxisBasic.LimitLoadReady;
  ax.Status.IsBrakeManuallyReleased := ax.fbMpAxisBasic.BrakeReleased;

  // Now load the sMot_AxisStatus structure with the data returned from the fb
  fctGetMpAxisInfo(_I_MpInfo := ADR(ax.fbMpAxisBasic.Info), _IO_UdtStatus := ax.Status);
  // further unpack diag info into fb status structure for easier access
  ax.statusFpMpAxisBasic.StatusId := ax.Status.AxisDiagnostics.StatusID.ID;
  ax.statusFpMpAxisBasic.StatusSeverity := ax.Status.AxisDiagnostics.StatusID.Severity;
  ax.statusFpMpAxisBasic.StatusCode := ax.Status.AxisDiagnostics.StatusID.Code;
  ax.statusFpMpAxisBasic.InternalId := ax.Status.AxisDiagnostics.Internal.ID;
  ax.statusFpMpAxisBasic.InternalSeverity := ax.Status.AxisDiagnostics.Internal.Severity;
  ax.statusFpMpAxisBasic.InternalFacility := ax.Status.AxisDiagnostics.Internal.Facility;
  ax.statusFpMpAxisBasic.InternalCode := ax.Status.AxisDiagnostics.Internal.Code;
  ax.statusFpMpAxisBasic.ExecutingCommand := ax.Status.AxisDiagnostics.ExecutingCommand;

  // Calculate special (algorithmic) positions
  CalcSpecialPositions;

  // Now that the status of this axis is known, copy it to the other axes slave status
  // area if this axis is specified as a slave.
  CopySlaveStatusToMaster;

END_ACTION

ACTION ActionMpAxisCoupling:
  // 1) Packs the sMot_CouplingParameters into a local axisCouplingParamsStructure
  // 2) Detects parameter changes and manages the Update and UpdateDone bits
  // 3) Sets the fb command bits based on the axis sMot_AxisCommands structure
  // 4) Runs the fbMpAxisCoupling funciton block
  // 5) Updates the axis structure with the status and axis info coming back from the fb

  // The execution behavior is determined by the inputs set elsewhere
  // in particular the sMot_AxisCommands Engage/Disengage Slave bits,
  // and the values in sMot_CouplingParameters struture.

  // Axis references set in init routine

  // Only enable the coupling fb if the axis number has been set,
  // the slave axis number has been set, and neither is set to be ignored.
  IF NOT ax.Ignore AND ax.AxisNo <> AD_UNKNOWN AND
     ax.CouplingParameters.SlaveAxisNo <> AD_UNKNOWN AND
     NOT axes[ax.CouplingParameters.SlaveAxisNo].Ignore THEN
    ax.fbMpAxisCoupling.Enable := TRUE;
  ELSE
    ax.fbMpAxisCoupling.Enable := FALSE;
  END_IF;

  // If the slave axis has changed, update the fb link to the slave axis
  // Handle this change before the call to fbUpdateCFbParams because
  // a slave number change would be detected but not handled by fbUpdateCFbParams.
  IF ax.CouplingParameters.SlaveAxisNo <> ax.CouplingParametersPrev.SlaveAxisNo THEN
    // Set the axis object based on the slave number
    IF ax.CouplingParameters.SlaveAxisNo <> AD_UNKNOWN THEN
      ax.SlaveAxisObj := axes[ax.CouplingParameters.SlaveAxisNo].AxisObj;
    ELSE
      ax.SlaveAxisObj := axDummySlave;
    END_IF;
    ax.fbMpAxisCoupling.MpLink := ADR(ax.SlaveAxisObj);
    // Update the previous value now that the change is handled
    ax.CouplingParametersPrev.SlaveAxisNo := ax.CouplingParameters.SlaveAxisNo;
  END_IF;

  // Load the parameters from the sMot_CouplingParameters structure into
  // local structure variables used for the call to fbMpAxisCoupling
  fctPackMpAxisCouplingParams(_I_UdtParams:= ADR(ax.CouplingParameters), _IO_MpParams := axisCouplingParams);

  // To allow coupling parameter changes to take effect without having to stop,
  // detect a difference between the desired parameters and the previous values.
  // If they are different, then set the update bit until the UpdateDone bit is set.
  // NOTE: This fb manages the ax.fbMpAxisCoupling.Update request and monitors the .UpdateDone bit
  // Use the .UpdateCouplingParams bit in the command structure if the application needs to control
  // when to trigger the update. If parameters need to be set in possibly different areas of the software,
  // and all the updates should take place at once, the update fb is called conditionally. The
  // checked bit can be set high so it is called all the time if the checked bit is not managed.
  ax.Commands.UpdateCouplingParams:= TRUE;
  IF ax.CouplingParameters.SlaveAxisNo <> AD_UNKNOWN AND ax.Commands.UpdateCouplingParams THEN
    ax.fbUpdateCFbParams();
    ax.Commands.UpdateCouplingParams := FALSE;
  END_IF;

  // Use the commands from the axis structue
  ax.fbMpAxisCoupling.ErrorReset := ax.Commands.DriveResetCmd;

  // Gear in if there is a slave, it is requested and it is allowed by the slave
  ax.fbMpAxisCoupling.Gear := ax.CouplingParameters.SlaveAxisNo <> AD_UNKNOWN AND ax.CouplingParameters.GearInCmd AND axes[ax.CouplingParameters.SlaveAxisNo].CouplingParameters.CouplingPermissive;
  ax.fbMpAxisCoupling.Cam := FALSE; // Not using camming
  // Gear in position if there is a slave, it is requested and it is allowed by the slave
  ax.fbMpAxisCoupling.GearInPos := ax.CouplingParameters.SlaveAxisNo <> AD_UNKNOWN AND ax.CouplingParameters.GearInPosCmd AND axes[ax.CouplingParameters.SlaveAxisNo].CouplingParameters.CouplingPermissive;
  // Generate an offset or phase shift if there is a slave, it is requested and it is allowed by the slave
  ax.fbMpAxisCoupling.OffsetShift := ax.CouplingParameters.SlaveAxisNo <> AD_UNKNOWN AND ax.CouplingParameters.OffsetShiftCmd AND axes[ax.CouplingParameters.SlaveAxisNo].CouplingParameters.CouplingPermissive;
  ax.fbMpAxisCoupling.PhaseShift := ax.CouplingParameters.SlaveAxisNo <> AD_UNKNOWN AND ax.CouplingParameters.PhaseShiftCmd AND axes[ax.CouplingParameters.SlaveAxisNo].CouplingParameters.CouplingPermissive;
  ax.fbMpAxisCoupling.GetCamPosition := FALSE; // not using camming
  ax.fbMpAxisCoupling.CamPrepare := FALSE; // not using camming
  ax.fbMpAxisCoupling.Recovery := FALSE; // not using camming

  // Call the fb
  ax.fbMpAxisCoupling();

  // Update the fb status structure
  ax.statusFpMpAxisCoupling.Active := ax.fbMpAxisCoupling.Active;
  ax.statusFpMpAxisCoupling.Error := ax.fbMpAxisCoupling.Error;
  ax.statusFpMpAxisCoupling.StatusId := ax.fbMpAxisCoupling.StatusID;
  ax.statusFpMpAxisCoupling.UpdateDone := ax.fbMpAxisCoupling.UpdateDone;
  ax.statusFpMpAxisCoupling.CommandBusy := ax.fbMpAxisCoupling.CommandBusy;
  ax.statusFpMpAxisCoupling.CommandAborted := ax.fbMpAxisCoupling.CommandAborted;

  // Update the axis status structure
  ax.Status.IsCoordInCompensation := ax.fbMpAxisCoupling.InCompensation;
  ax.Status.IsCoordInSync := ax.fbMpAxisCoupling.InSync;
  ax.Status.IsCoordOffsetDone := ax.fbMpAxisCoupling.OffsetDone;
  ax.Status.IsCoordPhasingDone := ax.fbMpAxisCoupling.PhasingDone;
  ax.Status.IsCoordRecoveryDone := ax.fbMpAxisCoupling.RecoveryDone;

  // Now load the sMot_AxisStatus structure with the data returned from the fb
  fctGetMpCouplingInfo(_I_MpInfo := ADR(ax.fbMpAxisCoupling.Info), _IO_UdtStatus := ax.Status);
  // add to the isCoordSlaveReady status the slave coupling permissive
  ax.Status.IsCoordSlaveReady := ax.Status.IsCoordSlaveReady AND axes[ax.CouplingParameters.SlaveAxisNo].CouplingParameters.CouplingPermissive;
  // further unpack diag info into fb status structure for easier access
  ax.statusFpMpAxisCoupling.StatusId := ax.Status.CoordAxisDiagnostics.StatusID.ID;
  ax.statusFpMpAxisCoupling.StatusSeverity := ax.Status.CoordAxisDiagnostics.StatusID.Severity;
  ax.statusFpMpAxisCoupling.StatusCode := ax.Status.CoordAxisDiagnostics.StatusID.Code;
  ax.statusFpMpAxisCoupling.InternalId := ax.Status.CoordAxisDiagnostics.Internal.ID;
  ax.statusFpMpAxisCoupling.InternalSeverity := ax.Status.CoordAxisDiagnostics.Internal.Severity;
  ax.statusFpMpAxisCoupling.InternalFacility := ax.Status.CoordAxisDiagnostics.Internal.Facility;
  ax.statusFpMpAxisCoupling.InternalCode := ax.Status.CoordAxisDiagnostics.Internal.Code;
  ax.statusFpMpAxisCoupling.ExecutingCommand := ax.Status.CoordAxisDiagnostics.ExecutingCommand;

END_ACTION

ACTION CalcSpecialPositions :
  // If there is an algorithm needed for calculating a different position, it can be done here
  // If not, just use the axis position.

  // CalculatedPosition1
  // Calculate the inner position relative to the outer position, in degrees.
  // This assumes the zero/home position of both the Outer and Inner axes was set to zero when
  // the index lines are lined up with each other.
  // Calculated Position = Inner Pos - Outer Pos.
  // Make the result be +/- 180 degrees:
  // If I-O > 180 :  Calc Pos = Result - 360
  // If I-O < -180 : Calc Pos = Result + 360
  // The fctAziDiff function in GAMath library does this (pos A - pos B)

  IF NOT axes[AD_INNER_ECCENTRIC].Status.IsHomed OR NOT axes[AD_OUTER_ECCENTRIC].Status.IsHomed THEN
    // Inner and/or outer axis is not homed.
    // Use the sentinel value for the calculated positions.
    ax.Status.CalculatedPosition1 := INVALID_SENTINEL_REAL;
  ELSE
    // Both the inner and outer axes are referenced.
    // Calc the difference between them. I - O
    ax.Status.CalculatedPosition1 := fctAziDiff(
    _I_PosA :=  ax.Status.Position,
    _I_PosB := axes[AD_OUTER_ECCENTRIC].Status.Position);
  END_IF;

  ax.Status.CalculatedPosition2 := ax.Status.Position;
  ax.Status.CalculatedPosition3 := ax.Status.Position;

END_ACTION

ACTION CopySlaveStatusToMaster :
  // If this axis number is a slave to another axis, then copy this axis
  // status to the master axis structure. This is a convenience
  // so the HMI for example, only needs to look in one structure (the master) and
  // can access the slave status.

  // Loop thru the axes. If the axis of index has this axis specified as a slave axis,
  // copy this axis status to the axis of index slave status.
  // Axis 0 is a dummy axis, so it can be skipped.
  FOR axIdx := 1 TO AXIS_COUNT DO
    IF axes[axIdx].CouplingParameters.SlaveAxisNo = AXIS_NO THEN
      // This axis is a slave to the axis referenced by axIdx.
      // Copy this axis status to the indexed axis slave status
      fctCopyAxisStatus(_I_SrcStatus := ADR(ax.Status), _I_DestStatus := ADR(axes[axIdx].StatusSlave));
    END_IF;
  END_FOR;
END_ACTION
```

- ActionMotionFbs.st.bak (not shown)
